// TIA Portal V15 export
// export: Created 2018-05-29T12:25:38.1552518Z, ExportSetting WithDefaults, DisplayName Totally Integrated Automation Portal, DisplayVersion V15, DisplayName TIA Portal Openness, DisplayVersion V15, DisplayName STEP 7 Professional, DisplayVersion V15, DisplayName WinCC Professional, DisplayVersion V15
FUNCTION "phase_1_fc" : Void   // FC1, STL
TITLE = _fc
{ S7_Optimized_Access := 'TRUE' }
VERSION : 0.1
// First instance of fds_example test
// stored: AutoNumber true, UDAEnableTagReadback false
BEGIN

NETWORK
TITLE = Main
// comment: First instance of fds_example
// Call the EM FB with the corresponding DB instance
CALL phase_example, phase_1
	EM_I_OUT_ID := 
	XV003_OPN := XV300.QOPEN
	XV003_CLS := XV300.QCLOSE
	XV003_MERR := XV300.QMON_ERR
	XV004_OPN := XV400.QOPEN
	XV004_CLS := XV400.QCLOSE
	XV004_MERR := XV400.QMON_ERR
	XV005_OPN := XV500.QOPEN
	XV005_CLS := XV500.QCLOSE
	XV005_MERR := XV500.QMON_ERR
	P001_RUN := P100.QRUN
	P001_STOP := P100.QSTOP
	P001_MERR := P100.QMON_ERR
	P001_MPS := P100.QMPS
	P002_RUN := P200.QRUN
	P002_STOP := P200.QSTOP
	P002_MERR := P200.QMON_ERR
	P002_MPS := P200.QMPS
	LT001_PV := LT100.QfVal
	LT001_AHH := LT100.LIM_Qb01
	LT001_AH := LT100.LIM_Qb02
	LT001_AL := LT100.LIM_Qb03
	LT001_ALL := LT100.LIM_Qb04
	LT001_ERR := LT100.QERR
	LT002_PV := LT200.QfVal
	LT002_AHH := LT200.LIM_Qb01
	LT002_AH := LT200.LIM_Qb02
	LT002_AL := LT200.LIM_Qb03
	LT002_ALL := LT200.LIM_Qb04
	LT002_ERR := LT200.QERR
	FIC001_PV := FIC100.PV
	FIC001_ERR := FIC100.QERR
	XV003_CMD := XV300.AUT_OP
	XV004_CMD := XV400.AUT_OP
	XV005_CMD := XV500.AUT_OP
	P001_ON := P100.AUTO_ON
	P001_AUT := P100.L_AUT
	P002_ON := P200.AUTO_ON
	P002_AUT := P200.L_AUT
	FIC001_EXT := FIC100.L_REMOTE
	FIC001_SP := FIC100.HMI_SP_INT
	FIC001_AUT := FIC100.L_AUT
	FIC001_VAL_OUT := FIC100.HMI_MAN
	FIC001_SET_SP := FIC100.Set_SP
	FIC001_SET_OUT := FIC100.Set_Output
END_FUNCTION
